{attribute 'no_check'}
FUNCTION_BLOCK AnalogIn
VAR_INPUT
	MinValue												: 	LREAL 	:= 0.0; //In case of extended range (107%), set Options.5 or MinValue accordingly e.g. -10.7V (instead of -10.0V as scaling is based on full 16bit)
	MaxValue												: 	LREAL 	:= 0.0; //In case of extended range (107%), set Options.5 or MaxValue accordingly e.g. 10.7V (instead of 10.0V as scaling is based on full 16bit)
	NoOfDigits												: 	INT 	(0..10)	:= 0; 	//number of decimal digits of scaled Q variable 
	OutOnError												:	LREAL 	:= 0.000000000000000001;
{attribute 'displaymode':='binary'}                     	
	Options													:	BYTE  := 2#0000_0000; (* 	.0 = FALSE scale value from 0 <-> 32767 / TRUE scale value with sign -32768 <-> 32767
																							.4 = Active only if .0 AND .5 =TRUE | FALSE scale value min -32768 / TRUE scale value changed from -30518 to -7629 -> Ext. Range Mode of e.g. 4-20mA where 0mA is equel -7629 
																							.5 = FALSE legacy range with FSV OF 100%=+-32767 / TRUE TO enable extended range AND applying ~7% TO MIN/MaxValue (with ext. range act. measurement can be exceeded OR undershot BY approx. 7% setting FSV TO 100%=+/-30518 AND 107% representing full 16BIT) 
																							For Scaling of 4-20mA according to NAMUR bit .0,.4 and .5 have to be set *)

																							
	Offset													:	LREAL := 0.0;
END_VAR                 									
VAR                                                     	
END_VAR                                                 	
VAR_OUTPUT                                              	
	Q														:	LREAL;		//Scaled result value
	In											AT  %I* 	: 	INT; 		//Hardware Input

{attribute 'displaymode':='binary'}                     	
	Status										AT  %I*		:	WORD := 2#0000_0000_0000_0000; //Terminal status word -> can also be linked with status byte 
END_VAR
VAR
END_VAR

(* read analog value 																					   *)
(* resolution process image			e.g.							/ 0V = 0 / 10V = 32767 / -10V = -32768 *)
(* or directly with NoOfDigits																	250 -> 25.0°*)
(************************************************************************************************************)
	
(* Scaling ******************************************************************)
	IF MaxValue <> MinValue 
	THEN
		Q 													:= Offset + scale2(In , SEL(Options.0, 0.0, SEL(Options.5 , -32768.0, SEL(Options.4, -30518.0,-7629.0) ) ), SEL(Options.5,32767.0,30518.0), MinValue, MaxValue);
		IF NoOfDigits > 0
		THEN
			Q												:= TO_FMLREAL(Q,NoOfDigits);
		END_IF
	
	ELSIF NoOfDigits > 0 (* Bsp PT100 *)
	THEN
		Q													:= Offset + TO_FMLREAL(In,NoOfDigits);
		
	ELSE  													
		Q 													:= 0.0;
	END_IF

	IF 	Error AND OutOnError <> 0.000000000000000001
	THEN
		Q													:= OutOnError;
	END_IF
(**********************************************************************************************************************)

{attribute 'monitoring' := 'call'}
PROPERTY PUBLIC Error : BOOL
GET
Error					:= Status.6 OR MinValue = MaxValue AND NoOfDigits = 0;
END_GET
END_PROPERTY

{attribute 'monitoring' := 'call'}
PROPERTY PUBLIC Limit_1 : BYTE
GET
Limit_1.0					:= Status.2;
Limit_1.1					:= Status.3;
END_GET
END_PROPERTY

{attribute 'monitoring' := 'call'}
PROPERTY PUBLIC Limit_2 : BYTE
GET
Limit_2.0					:= Status.4;
Limit_2.1					:= Status.5;
END_GET
END_PROPERTY

PROPERTY PUBLIC optEnableScaleExtRangeMode : bool
GET
optEnableScaleExtRangeMode := Options.5;
END_GET
SET
Options.5 := optEnableScaleExtRangeMode;
END_SET
END_PROPERTY

PROPERTY PUBLIC optEnableScaleExtRangeModeNeg7629 : bool
GET
optEnableScaleExtRangeModeNeg7629 := Options.4;
END_GET
SET
Options.4 := optEnableScaleExtRangeModeNeg7629;
END_SET
END_PROPERTY

PROPERTY PUBLIC optEnableScaleSignedValue : bool
GET
optEnableScaleSignedValue := Options.0;
END_GET
SET
Options.0 := optEnableScaleSignedValue;
END_SET
END_PROPERTY

{attribute 'monitoring' := 'call'}
PROPERTY PUBLIC Overrange : BOOL
GET
Overrange					:= Status.1;
END_GET
END_PROPERTY

{attribute 'monitoring' := 'call'}
PROPERTY PUBLIC SyncError : BOOL
GET
SyncError 			:= Status.13;
END_GET
END_PROPERTY

{attribute 'monitoring' := 'call'}
PROPERTY PUBLIC TxPDOState : BOOL
GET
TxPDOState					:= Status.14; //True if not valid
END_GET
END_PROPERTY

{attribute 'monitoring' := 'call'}
PROPERTY PUBLIC TxPDOToggle : BOOL
GET
TxPDOToggle						:= Status.15;
END_GET
END_PROPERTY

{attribute 'monitoring' := 'call'}
PROPERTY PUBLIC Underrange : BOOL
GET
Underrange 					:= Status.0;
END_GET
END_PROPERTY

END_FUNCTION_BLOCK

(* stored: Version 1.1.0.1, ProductVersion 3.1.4024.15
   POU AnalogIn: Id {dde11646-3149-4a70-b74f-55d9fab28ad0}, SpecialFunc None
   Property Error: Id {31470864-20ca-4d53-a541-6c9ddff36cc3}
   Get Get: Id {4098ce75-4c4f-4cc1-924c-86477941e2de}
   Property Limit_1: Id {20c7498c-260b-4a27-9ceb-0974490d21d5}
   Get Get: Id {32e3b45e-ff85-45f1-906c-ba0848ebbf4a}
   Property Limit_2: Id {a9cc8e21-4a81-40db-aea3-c10633c8dbcd}
   Get Get: Id {15ae6286-32ee-499c-b9fd-5184d9fc1100}
   Property optEnableScaleExtRangeMode: Id {f80202c2-77b7-4301-9c72-35cdec25263c}
   Get Get: Id {ebb26774-963d-41fe-91b1-3ae35adc73cb}
   Set Set: Id {63bab101-2643-4b9a-975e-012fb0869c58}
   Property optEnableScaleExtRangeModeNeg7629: Id {e113c5fa-63ef-4144-9754-635bbae9d06c}
   Get Get: Id {9b0248cb-7f26-4888-9d79-5dccc4b67361}
   Set Set: Id {1476a9f2-aa27-4f4d-b934-769c0dfe1bee}
   Property optEnableScaleSignedValue: Id {3d04c02d-caa5-4b6b-9c84-63c0a3f425e9}
   Get Get: Id {19f6e4ac-7636-407b-a83a-99210f706653}
   Set Set: Id {6472af38-88de-45a1-9991-a49c9740a648}
   Property Overrange: Id {a8762b0c-16e0-4662-8619-04f76f8daee4}
   Get Get: Id {6c692a07-01c1-4499-9f0d-3f93de54c08c}
   Property SyncError: Id {7a3100ac-d584-4529-b93f-cd3cb78cd5b0}
   Get Get: Id {d7b4720f-e2ad-499d-a202-d3f7a3c502c5}
   Property TxPDOState: Id {0d144e83-ae62-46b5-828d-274ae6f36b07}
   Get Get: Id {a3a57494-bfc2-4925-ac1f-90a64d5660c4}
   Property TxPDOToggle: Id {cad01e06-5fc5-49c6-bb1e-e71e8e4e51a2}
   Get Get: Id {9d210938-627d-440f-bc44-b9e7c30e6e13}
   Property Underrange: Id {0ede74a4-9635-4354-99e2-58892ae26e7f}
   Get Get: Id {49227475-056d-4dfc-85d5-3df4995e9f7a} *)
